{attribute 'linkalways'} 
{attribute 'no_explicit_call' := 'This FB is a CLASS and must be accessed using methods or properties'}
{attribute 'enable_dynamic_creation'}
FUNCTION_BLOCK FINAL XOR_USINT EXTENDS Node
VAR
	in1 : _USINT(0);
	in2 : _USINT(0);
	out : _USINT(0);
END_VAR

METHOD PUBLIC Clone : I_Node
VAR
	pNode : POINTER TO XOR_USINT;
END_VAR
pNode := __NEW(XOR_USINT);
Clone := pNode^;
END_METHOD

METHOD FB_init : BOOL
VAR_INPUT
	bInitRetains : BOOL; // if TRUE, the retain variables are initialized (warm start / cold start)
	bInCopyCode : BOOL;  // if TRUE, the instance afterwards gets moved into the copy code (online change)
END_VAR
AddInput('in1',THIS^.in1);
AddInput('in2',THIS^.in2);
AddOutput('out', THIS^.out);
END_METHOD

METHOD PROTECTED OnExecute
VAR
END_VAR
out.Value := in1.Value XOR in2.Value;
END_METHOD

END_FUNCTION_BLOCK

(* stored: Version 1.1.0.1, ProductVersion 3.1.4024.15
   POU XOR_USINT: Id {8138ce4d-0b21-4163-b065-2825f879c5ec}, SpecialFunc None
   Folder Constructor: Id {5ebb8aa8-028f-4091-990f-dbecf4d63811}
   Method Clone: Id {866d068b-f7df-4100-aa2d-53408478ff22}
   Method FB_init: Id {f4b85cf8-ec2a-43a1-b084-112e771a1962}
   Method OnExecute: Id {4f8cf86d-494f-4407-a91f-4630f8c63f1a} *)
